TYPE XTSMainStatus_typ :
STRUCT
	State	: XTSMainState_enum;
END_STRUCT
END_TYPE

(* stored: Version 1.1.0.1, ProductVersion 3.1.4024.12
   DUT XTSMainStatus_typ: Id {acd24958-713c-06a0-049c-e092c76fb1c4} *)
